PROGRAM POU
VAR
	
	i : INT := 0;
	f : REAL := 0.0;
	elapsed : TIME := TIME#0M0S0MS;
	today : DATE := DATE#2020-01-01;
	message : STRING := '';
	count : BYTE := 0;
	
	A AT %I* : BOOL := FALSE;
	B AT %I* : BOOL := FALSE;
	C AT %I* : BOOL := FALSE;
	D AT %Q* : BOOL := FALSE;
		
	op1 : INT := 1;
	op2 : INT := 2;
	res : REAL := 0.0;
	test : BOOL := FALSE;
	
	TON_0: TON;
	
END_VAR

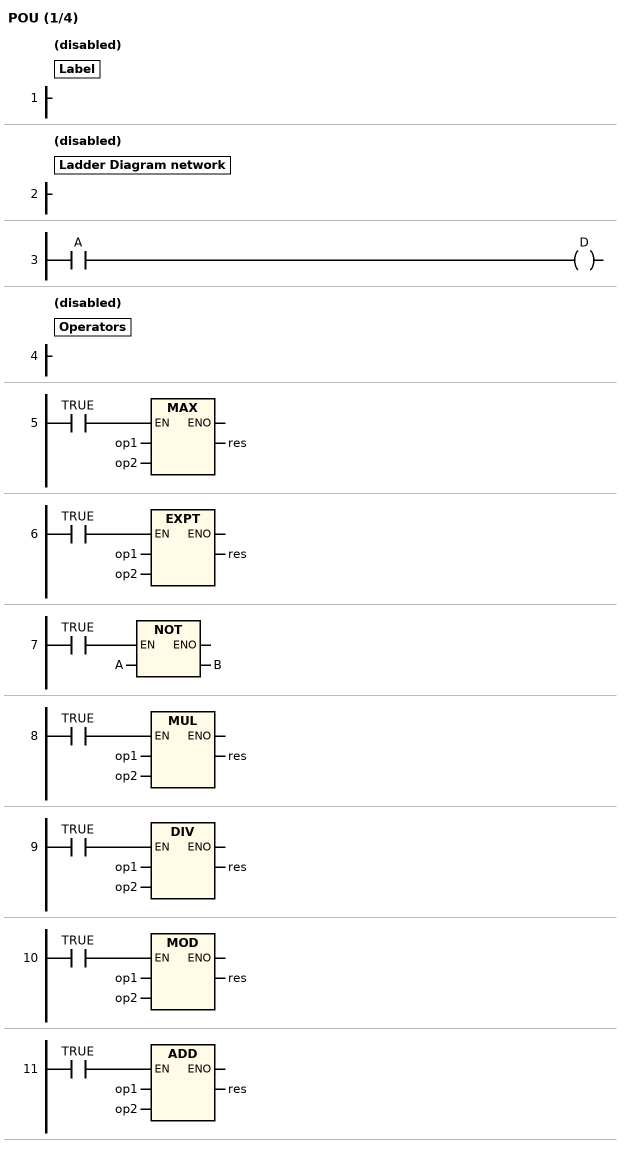
// NETWORK 1 (disabled)
// label: Label

// NETWORK 2 (disabled)
// label: Ladder Diagram network

// NETWORK 3
D := A;

// NETWORK 4 (disabled)
// label: Operators

// NETWORK 5
res := MAX(op1, op2);

// NETWORK 6
res := EXPT(op1, op2);

// NETWORK 7
B := NOT A;

// NETWORK 8
res := op1 * op2;

// NETWORK 9
res := op1 / op2;

// NETWORK 10
res := op1 MOD op2;

// NETWORK 11
res := op1 + op2;

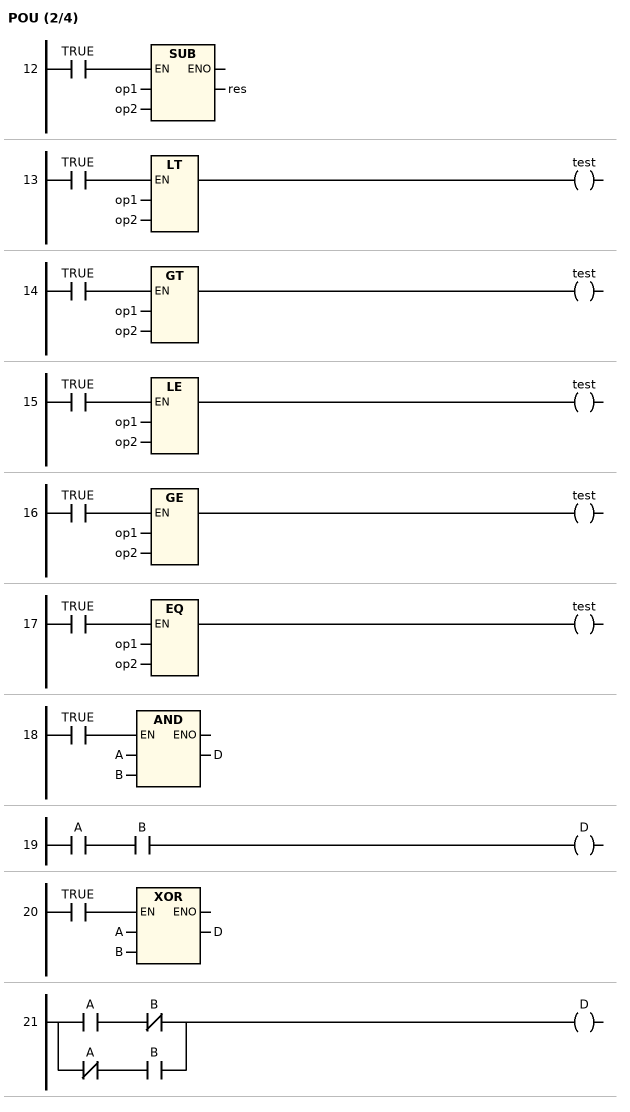
// NETWORK 12
res := op1 - op2;

// NETWORK 13
test := op1 < op2;

// NETWORK 14
test := op1 > op2;

// NETWORK 15
test := op1 <= op2;

// NETWORK 16
test := op1 >= op2;

// NETWORK 17
test := op1 = op2;

// NETWORK 18
D := A AND B;

// NETWORK 19
D := A AND B;

// NETWORK 20
D := A XOR B;

// NETWORK 21
D := A AND NOT B OR NOT A AND B;

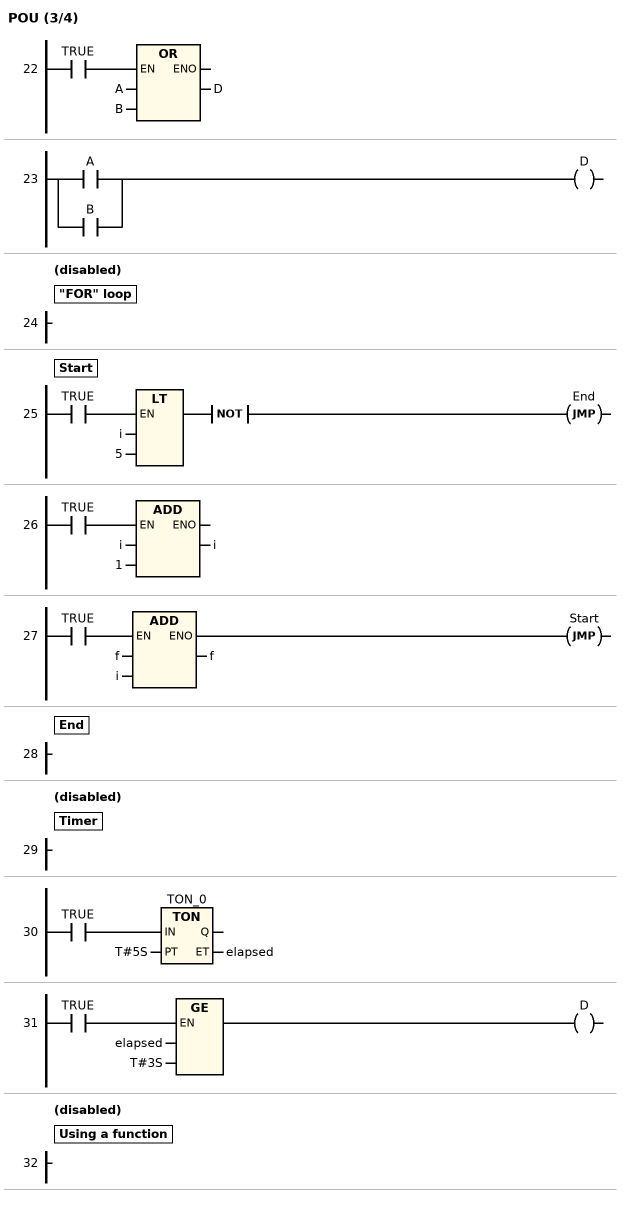
// NETWORK 22
D := A OR B;

// NETWORK 23
D := A OR B;

// NETWORK 24 (disabled)
// label: "FOR" loop

// NETWORK 25
Start:
IF NOT (i < 5) THEN JMP End; END_IF

// NETWORK 26
i := i + 1;

// NETWORK 27
f := f + i;
JMP Start;

// NETWORK 28
End: ;

// NETWORK 29 (disabled)
// label: Timer

// NETWORK 30
TON_0(IN := TRUE, PT := T#5S, ET => elapsed); // TON

// NETWORK 31
D := elapsed >= T#3S;

// NETWORK 32 (disabled)
// label: Using a function

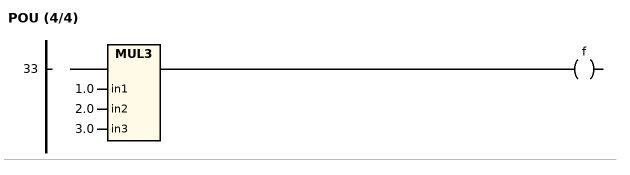
// NETWORK 33
f := MUL3(in1 := 1.0, in2 := 2.0, in3 := 3.0);

END_PROGRAM

(* stored: Version 1.1.0.1, ProductVersion 3.1.4024.3
   POU POU: Id {bf5de3b6-88ba-4c75-ae2e-f538a68bd75e}, SpecialFunc None *)
